Omron CX-Programmer project NewProject (CX-Programmer 9.50)

# PLC PLC_OMRON: CJ2M CPU11
; TEST 23/08/18

## Global symbols (name address type ; comment)
PB1 0.00 BOOL  ; PUSH BUTTON 1
RESET 0.01 BOOL  ; out1

## Program NewProgram1 (cyclic task 0)

### Section Section1

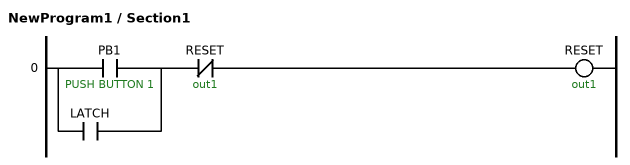
; rung 0
LD PB1  ; PUSH BUTTON 1
OR LATCH
ANDNOT RESET  ; out1
OUT RESET  ; out1

### Section END
; rung 0
END(001)